FUNCTION F_AlpacaFormatUri : STRING
VAR_INPUT
    sDeviceName     : STRING;
    nDeviceNumber   : UINT;
    sVariableName   : STRING;
END_VAR
VAR
END_VAR

F_AlpacaFormatUri := CONCAT('/api/v1/',
                     CONCAT(sDeviceName,
                     CONCAT('/',
                     CONCAT(UINT_TO_STRING(nDeviceNumber),
                     CONCAT('/', sVariableName)))));

END_FUNCTION

(* stored: Version 1.1.0.1, ProductVersion 3.1.4024.12
   POU F_AlpacaFormatUri: Id {8b2c565c-6e6e-40bd-99d2-d58fa09683cc}, SpecialFunc None *)
